//{attribute 'conditionalshow' := 'SomeText'}
//{attribute 'conditionalshow'}
//{attribute 'hide'}
VAR_GLOBAL CONSTANT
END_VAR

(* stored: Version 1.1.0.1, ProductVersion 3.1.4024.11
   GVL Constants: Id {1af09cf5-e05e-4d97-81aa-7dd3bf8f41b4} *)
